Staubli VAL3: handleLtype.pgx

program handleLtype(string& x_sItemSelected[])
  local num l_i
  local bool l_bQuit
  local num l_nKeyPressed
  local num l_nRow
  local num l_nCol
  local num l_nWidth
  local num l_nHeight
  local num l_nSizeOfList
  local num l_nIdx
  local string l_sCommand
  local string l_sListName
  local string l_sItemSelected
begin
  // Display the list object
  //
  // Input Param
  // none
  //
  // Output Param
  // x_sItemSelected  : Item selected by user in the list
  //
  // Comments:
  //
  // Created 21/02/08                              CCUR
  //--------------------------------------------------------------
  //Get position of the list on the screen
  if (mid(pw:sTxtBoxType[nFocused],1,0)=="L") or (mid(pw:sTxtBoxType[nFocused],1,0)=="l")
    call ut:extractPos(right(pw:sTxtBoxType[nFocused],len(pw:sTxtBoxType[nFocused])-1),";",l_nRow,l_nCol)
  endIf
  // Get width and height of the list to display
  // format of sTxtBoxType is Lww;xx;yy;zz so remove Lxx;yy;
  call ut:_decode(pw:sTxtBoxType[nFocused],l_sCommand,";",0)
  call ut:_decode(l_sCommand,l_sCommand,";",0)
  call ut:extractPos(l_sCommand,";",l_nWidth,l_nHeight)
  l_nWidth=max(5,l_nWidth)
  l_nHeight=max(2,l_nHeight)
  //
  l_sListName="pw:sListItem"+toString("",nFocused)
  resize(sListItems,1,pw:nListSize[nFocused])
  //
  if getData(l_sListName,sListItems)>0
    // Create the list of items
    call up:listSetSize(l_nCol,l_nRow,l_nWidth,l_nHeight)
    call up:listCreate("ItemList")
    call up:listAdd(sListItems)
    // Display list of items
    call up:listUpdate(0)
    //
    // EVENT LOOP
    l_bQuit=false
    do
      l_nKeyPressed=getKey()
      call up:listEvent(l_nKeyPressed,l_nIdx,l_sItemSelected)
      switch l_nKeyPressed
        // Return
        case 270
          x_sItemSelected=l_sItemSelected
          l_bQuit=true
        break
        // Escape
        case 255
          l_bQuit=true
        break
      endSwitch
    until l_bQuit
  else
    // Error code please !!!
  endIf
end
